// TIA Portal V20 export
// export: Created 2025-12-01T14:57:18.1741148Z, ExportSetting None, DisplayName Totally Integrated Automation Portal, DisplayVersion V20 Update 3, DisplayName TIA Portal Openness, DisplayVersion V20 Update 3, DisplayName TIA Portal Version Control Interface, DisplayVersion V20 Update 3, DisplayName STEP 7 Professional, DisplayVersion V20 Update 3, DisplayName STEP 7 Safety, DisplayVersion V20 Update 2, DisplayName WinCC Basic/Comfort/Advanced, DisplayVersion V20 Update 3, DisplayName WinCC Professional, DisplayVersion V20 Update 3, DisplayName WinCC Unified, DisplayVersion V20 Update 3
DATA_BLOCK "DB839_DispositivosVarios"   // DB839
{ S7_Optimized_Access := 'FALSE' }
AUTHOR : TRACKING
NAME : 20160411
VERSION : 3.1
// stored: AutoNumber false
   VAR
      DispoBaliza { S7_SetPoint := 'True'} : Array[0.."CTE_MaxDispositivosBaliza"] of "UDT_DatosBaliza";   // Datos del Dispositivo Baliza
      DispoLlave { S7_SetPoint := 'True'} : Array[0.."CTE_MaxDispositivosLlave"] of "UDT_DatosLlave";   // Datos del Dispositivo Llave
      DispoSeta { S7_SetPoint := 'True'} : Array[0.."CTE_MaxDispositivosSeta"] of "UDT_DatosSeta";   // Datos del Dispositivo Seta
      DispoBarrera { S7_SetPoint := 'True'} : Array[0.."CTE_MaxDispositivosBarrera"] of "UDT_DatosBarrera";   // Datos del Dispositivo Barrera
      DispoPuerta { S7_SetPoint := 'True'} : Array[0.."CTE_MaxDispositivosPuerta"] of "UDT_DatosPuerta";   // Datos del Dispositivo Puerta
      DispoLineaPotencia { S7_SetPoint := 'True'} : Array[0.."CTE_MaxDispositivosLineaPotencia"] of "UDT_DatosLineaPotencia";   // Datos del Dispositivo Linea de Potencia
   END_VAR
BEGIN
END_DATA_BLOCK
